// TIA Portal V17 export
// export: Created 2023-07-20T16:54:10.2633387Z, ExportSetting WithDefaults, DisplayName Totally Integrated Automation Portal, DisplayVersion V17, DisplayName TIA Portal Openness, DisplayVersion V17, DisplayName TIA Portal Version Control Interface, DisplayVersion V17, DisplayName STEP 7 Professional, DisplayVersion V17, DisplayName STEP 7 Safety, DisplayVersion V17, DisplayName WinCC Professional, DisplayVersion V17
FUNCTION "Valves" : Void   // FC1050, FBD
{ S7_Optimized_Access := 'TRUE' }
VERSION : 0.1
// stored: AutoNumber false, IsIECCheckEnabled false, SetENOAutomatically false, UDAEnableTagReadback false
   VAR_INPUT
      "Motion enable" : Bool;
      Trigger : Bool;
      "Auto mode" : Bool;
      "Manual mode" : Bool;
      "HMI S12" : Bool;
      "HMI S14" : Bool;
      "S12 sensors" : Bool;
      "S14 sensors" : Bool;
      "S12 motion time" : Time;
      "S14 motion time" : Time;
   END_VAR
   VAR_OUTPUT
      S12 : Bool;
      S14 : Bool;
      "Alarm motion code" : USInt;
   END_VAR
   VAR_IN_OUT
      "S12 motion timer" : TON_TIME;
      "S14 motion timer" : TON_TIME;
   END_VAR
   VAR_TEMP
      "temp S12" : Bool;
      "temp S14" : Bool;
      "temp S12 motion fault" : Bool;
      "temp S14 motion fault" : Bool;
   END_VAR
   VAR_TEMP   // added for the SCL form of the ladder/FBD networks
      _w1 : Bool;
   END_VAR
BEGIN

REGION Network 1: Control logic
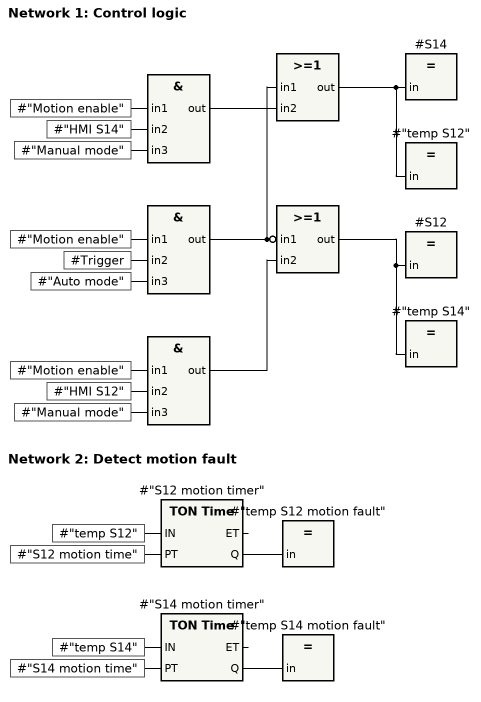
   #_w1 := #"Motion enable" AND #Trigger AND #"Auto mode";
   #S14 := #_w1 OR (#"Motion enable" AND #"HMI S14" AND #"Manual mode");
   #"temp S12" := #S14;
   #S12 := NOT #_w1 OR (#"Motion enable" AND #"HMI S12" AND #"Manual mode");
   #"temp S14" := #S12;
END_REGION

REGION Network 2: Detect motion fault
   #"S12 motion timer"(IN := #"temp S12", PT := #"S12 motion time");   // TON
   #"temp S12 motion fault" := #"S12 motion timer".Q;
   #"S14 motion timer"(IN := #"temp S14", PT := #"S14 motion time");   // TON
   #"temp S14 motion fault" := #"S14 motion timer".Q;
END_REGION

REGION Network 3: Motion alarms
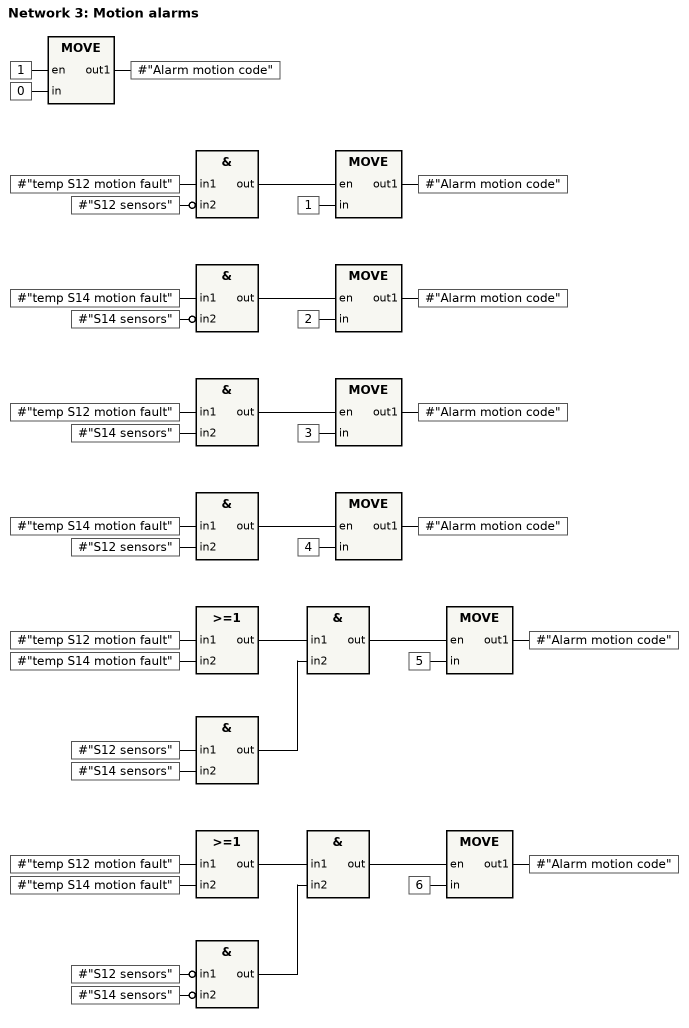
   IF 1 THEN #"Alarm motion code" := 0; END_IF;
   IF #"temp S12 motion fault" AND NOT #"S12 sensors" THEN #"Alarm motion code" := 1; END_IF;
   IF #"temp S14 motion fault" AND NOT #"S14 sensors" THEN #"Alarm motion code" := 2; END_IF;
   IF #"temp S12 motion fault" AND #"S14 sensors" THEN #"Alarm motion code" := 3; END_IF;
   IF #"temp S14 motion fault" AND #"S12 sensors" THEN #"Alarm motion code" := 4; END_IF;
   IF (#"temp S12 motion fault" OR #"temp S14 motion fault") AND #"S12 sensors" AND #"S14 sensors" THEN
       #"Alarm motion code" := 5;
   END_IF;
   IF (#"temp S12 motion fault" OR #"temp S14 motion fault") AND NOT #"S12 sensors" AND NOT #"S14 sensors" THEN
       #"Alarm motion code" := 6;
   END_IF;
END_REGION
END_FUNCTION
